PROGRAM MAIN
VAR
	nCount : UDINT;
	tBlink :TON;       // timer instance -it has its own memory
	bLight : BOOL;     // the output that will blink
END_VAR

nCount := nCount + 1;

// run the timer; when it expires, toggle the light and restart
tBlink(IN := NOT tBlink.Q, PT := T#500MS);

IF tBlink.Q THEN
	bLight := NOT bLight;
END_IF

GVL_ModbusIO.mwActuators.0 := bLight;
GVL.mb_Output_Registers[0].0 := bLight;

END_PROGRAM

(* stored: Version 1.1.0.1, ProductVersion 3.1.4026.18
   POU MAIN: Id {055f7781-fa15-44cb-9bbe-9f4c327b774f}, SpecialFunc None *)
